// TIA Portal V20 export
TYPE "typeCmControlNode"
// stored: Namespace Unit1.Em4
   STRUCT
      Interlock { ExternalWritable := 'False'} : "Unit1.Em4.typeCmControlNodeInterlock";
      softcam { ExternalWritable := 'False'} : "Unit1.Em4.typeCmControlNodeSoftCam";
      brakeTest { ExternalWritable := 'False'} : "Unit1.Em4.typeCmControlNodeBrakeTest";
   END_STRUCT;
END_TYPE
